TYPE timer_location:
    (Idle_timer_location, Running_timer_location);
END_TYPE

(* stored: ProductVersion 3.1.0.18, Version 1.1.0.1 *)
